FUNCTION_BLOCK FB_Homing_StandardNC EXTENDS FB_CyclicFB IMPLEMENTS I_MotionSequence
VAR
	_Axis : I_BasicAxis;
	fbMcHome : MC_Home;
	
	_bBusy, _bDone, _bError :BOOL;
	_bErrorID :UDINT;
	
	nStep :INT;
	
END_VAR

METHOD Abort
VAR_INPUT
END_VAR
fbMcHome(Axis := _Axis.Axis, Execute := FALSE);
_bBusy := FALSE;
nStep := 0;
END_METHOD


PROPERTY Axis : SPT_Motion_Control.I_BasicAxis
GET
Axis := _Axis;
END_GET
SET
_Axis := Axis;
END_SET
END_PROPERTY


PROPERTY Busy : BOOL
GET
Busy := _bBusy;
END_GET
END_PROPERTY


METHOD CyclicLogic
CASE nStep OF
    0: // IDLE
        fbMcHome(Axis := _Axis.Axis, Execute := FALSE);

    10: // TRIGGER HOMING
        fbMcHome(
            Axis        := _Axis.Axis, 
            Execute     := TRUE, 
            HomingMode  := MC_DefaultHoming, // <--- CZYTAJ Z PARAMETRÓW NC!
            bCalibrationCam := FALSE // Tutaj można podpiąć wejście, jeśli nie jest zlinkowane w NC
        );
        
        // Czekamy aż blok przyjmie komendę
        IF fbMcHome.Busy THEN
            nStep := 20;
        ELSIF fbMcHome.Error THEN
            nStep := 99;
        END_IF

    20: // WAIT FOR DONE
        // Wywołanie cykliczne
        fbMcHome(Axis := _Axis.Axis);
        
        IF fbMcHome.Done THEN
            _bBusy := FALSE;
            _bDone := TRUE;
            nStep := 0; // Koniec sukcesem
        ELSIF fbMcHome.Error THEN
            nStep := 99;
        END_IF

    99: // ERROR HANDLING
        _bBusy    := FALSE;
        _bError   := TRUE;
        _bErrorID := fbMcHome.ErrorID;
        nStep    := 0;
END_CASE
END_METHOD

PROPERTY Done : BOOL
GET
Done := _bDone;
END_GET
END_PROPERTY

PROPERTY Error : BOOL
GET
Error := _bError;
END_GET
END_PROPERTY

PROPERTY ErrorID : UDINT
GET
ErrorID := _bErrorID;
END_GET
END_PROPERTY


METHOD Execute : BOOL
// Reset i start
IF _Axis = 0 THEN RETURN; END_IF

_bBusy       := TRUE;
_bDone       := FALSE;
_bError      := FALSE;
_bErrorID    := 0;
nStep       := 10; // Start sekwencji
END_METHOD

PROPERTY InitComplete : BOOL
GET
END_GET
END_PROPERTY

END_FUNCTION_BLOCK

(* stored: Version 1.1.0.1, ProductVersion 3.1.4024.15
   POU FB_Homing_StandardNC: Id {a68036c7-0906-4add-a8ec-d72fc1d336c0}, SpecialFunc None
   Method Abort: Id {771dc933-2c39-43b9-9ff8-76313dbd940b}
   Property Axis: Id {33e35a1f-2c3a-4bfc-bb60-bae2383b8b6a}
   Get Get: Id {9ab12adb-c510-4298-96a4-7ffd2581d5f0}
   Set Set: Id {f767de7a-c1ca-4f02-9738-024b1923a2d6}
   Property Busy: Id {3753885d-a220-4799-8eac-648e681e4eb9}
   Get Get: Id {9fbfda9d-4904-4f9f-af47-7c558ece42f7}
   Method CyclicLogic: Id {3ee0a176-f137-4cd7-8aa9-6d46284035d2}
   Property Done: Id {9532d168-c50e-4321-997d-12356c697dc4}
   Get Get: Id {7e511263-a7b0-4b27-955f-f0a16a22967b}
   Property Error: Id {2ddf9516-adeb-45ba-822f-111669b0c9f8}
   Get Get: Id {3b22b156-3aae-4113-bcf9-ab311e7522b3}
   Property ErrorID: Id {08ec2b8b-d1ff-44e7-afef-4ed219024905}
   Get Get: Id {cbcd4fa1-fdf1-4329-aec3-52e3cfc72aa6}
   Method Execute: Id {0ce6e478-7e33-4c23-994a-236e753a0719}
   Property InitComplete: Id {adc32464-ccda-44e3-9865-b1afc471c266}
   Get Get: Id {d4f7d374-0999-4a2e-a160-1af9fa417971} *)
